{attribute addProperty BoxType "EP1122-0001-0017"}
{attribute addProperty Id "A_0026_EP1122_0001_0018A_0026_EP1122_0001_0018_C0E430961014268719478003.75"}
{attribute addProperty CRC "45315985"}
{attribute addProperty SizeInBites "10142"}
{attribute addProperty SizeInBytes "68719478003.75"}
TYPE A_0025_EP1122_0001_0017_02B37791 EXTENDS EP1122_179A0949 :
STRUCT
	{attribute addProperty Name "A_0026_EP1122_0001_0018"}
	A_0026_EP1122_0001_0018 : A_0026_EP1122_0001_0018_C0E43096;
END_STRUCT
END_TYPE

(* stored: Version 1.2.0.0, ProductVersion 3.1.4024.9
   DUT A_0025_EP1122_0001_0017_02B37791: Id {bf5e9232-b197-4c61-8042-34c59a5d5b7a} *)
